// TwinCAT 3 PLC project plc_example_demo
// Title: lcls-plc-example-demo
// ProjectVersion: 1.0.0
// ProgramVersion: 3.1.4023.0
// libraries:
//   lcls-twincat-motion, * (SLAC)
//   Tc2_Standard, * (Beckhoff Automation GmbH)
//   Tc2_System, * (Beckhoff Automation GmbH)
//   Tc3_Module, * (Beckhoff Automation GmbH)
// project tree:
//   / PlcTask.TcTTO
//   Version/ Global_Version.TcGVL
//   POUs/ MAIN.TcPOU
// real-time tasks:
//   TASK PlcTask: cycle T#10ms, priority 20, ADS port 350
// motion (NC):
// I/O:
//   DEVICE Device 1 (EtherCAT), AmsNetId 172.21.148.148.2.1
//     Term 1 (EK1200) [EK1200-5000 EtherCAT Power supply (2A E-Bus)]
//       Term 2 (EL7031)
//       Term 3 (EL5042) [EL5042 2Ch. BiSS-C Encoder]
//       Term 4 (EL3002) [EL3002 2Ch. Ana. Input +/-10V]
//       Term 5 (EL9011)
// variable links:
//   plc_example_demo Instance <-> Device 1 (EtherCAT)/Term 1 (EK1200)/Term 3 (EL5042)
//     PlcTask Inputs/MAIN.nEncoderCount <-> FB Inputs Channel 1/Position

CONFIGURATION plc_example_demo
    RESOURCE PLC ON TwinCAT3
        TASK PlcTask(INTERVAL := T#10ms, PRIORITY := 20);
        PROGRAM MAIN WITH PlcTask : MAIN;
    END_RESOURCE
END_CONFIGURATION

// ---- Version/Global_Version.TcGVL
{attribute 'TcGenerated'}
// This function has been automatically generated from the project information.
VAR_GLOBAL CONSTANT
    {attribute 'const_non_replaced'}
    {attribute 'linkalways'}
    stLibVersion_lcls_plc_example_demo : ST_LibVersion := (iMajor := 1, iMinor := 0, iBuild := 0, iRevision := 0, sVersion := '1.0.0');
END_VAR

// ---- POUs/MAIN.TcPOU
PROGRAM MAIN
VAR
    {attribute 'pytmc' := '
        pv: @(PREFIX):DEMO:COUNTER
        io: i
    '}
    nCounter: UDINT := 100;
    sError: STRING;

    {attribute 'TcLinkTo' := 'TIIB[Term 3 (EL5042)]^FB Inputs Channel 1^Position'}
    nEncoderCount AT %I*: ULINT;
    {attribute 'TcLinkTo' := 'TIIB[Term 6 (EL2004)]^Channel 1^Output'}
    bOutput AT %Q*: BOOL;
END_VAR

sError := F_MotionErrorCodeLookup(nCounter);
bOutput := TRUE;
IF sError = F_MotionErrorCodeLookup(1) THEN
    nCounter := nCounter + 2;
END_IF

END_PROGRAM
